FUNCTION_BLOCK F_ABS (* absolute value *)
  (* Standard: 61131-3; Classification: standard function of one numeric variable *)
  (* Version 0.0, 2013-04-24, 4DIAC-IDE, 4DIAC-Consortium *)
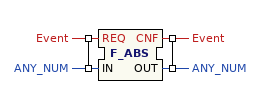
  EVENT_INPUT
    REQ WITH IN; (* Service Request *)
  END_EVENT
  EVENT_OUTPUT
    CNF WITH OUT; (* Confirmation of Requested Service *)
  END_EVENT
  VAR_INPUT
    IN : ANY_NUM; (* Event Input Qualifier *)
  END_VAR
  VAR_OUTPUT
    OUT : ANY_NUM; (* Event Output Qualifier *)
  END_VAR
END_FUNCTION_BLOCK
